(* CODESYS project traffic lights.project

Project tree, tasks and I/O mapping:
  Device : CODESYS Control Win V3, 3S - Smart Software Solutions GmbH, order no. 305021, version 3.5.7.0
    application Application
      libraries: Standard, * (System)
      task MainTask (cyclic, interval t#20ms, priority 1) calls PLC_PRG
      task VISU_TASK (cyclic, interval 100 ms, priority 31) calls VisuElems.Visu_Prg
      program PLC_PRG [LD]
      visualisation Visualization
  text list GlobalTextList
*)

// Device/Application/PLC_PRG
PROGRAM PLC_PRG

VAR
	TON_01: TON;
	t1: TIME;
	TP_01: TP;
	t11: TIME;
	F_TRIG_02: F_TRIG;
	TON_02: TON;
	t2: TIME;
	TP_02: TP;
	t22: TIME;
	F_TRIG_03: F_TRIG;
	F_TRIG_04: F_TRIG;
	TP_03: TP;
	TP_04: TP;
	t3: TIME;
	start: BOOL;
	stop: BOOL;
	lamp4: BOOL;
	lamp1: BOOL;
	lamp2: BOOL;
	lamp3: BOOL;
	red: BOOL;
	green: BOOL;
	amber: BOOL;
END_VAR

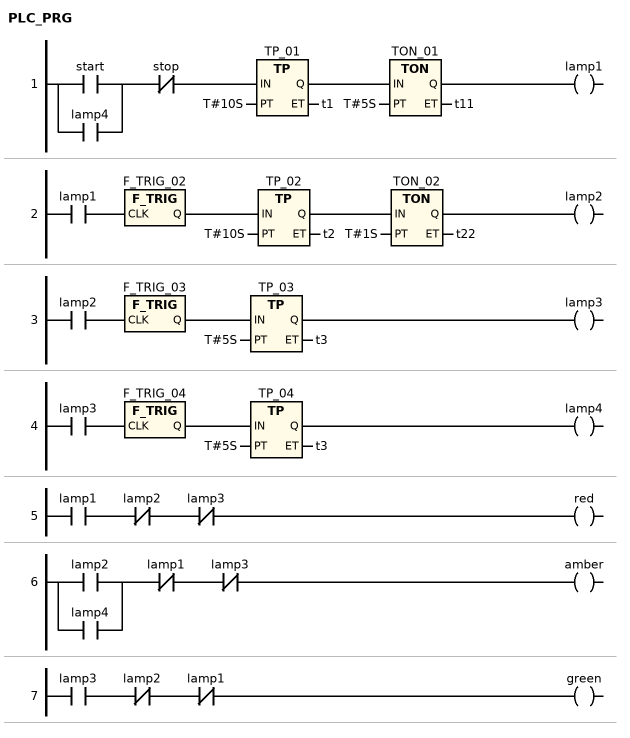
// NETWORK 1
TP_01(IN := (start OR lamp4) AND NOT stop, PT := T#10S, ET => t1); // TP
TON_01(IN := TP_01.Q, PT := T#5S, ET => t11); // TON
lamp1 := TON_01.Q;

// NETWORK 2
F_TRIG_02(CLK := lamp1); // F_TRIG
TP_02(IN := F_TRIG_02.Q, PT := T#10S, ET => t2); // TP
TON_02(IN := TP_02.Q, PT := T#1S, ET => t22); // TON
lamp2 := TON_02.Q;

// NETWORK 3
F_TRIG_03(CLK := lamp2); // F_TRIG
TP_03(IN := F_TRIG_03.Q, PT := T#5S, ET => t3); // TP
lamp3 := TP_03.Q;

// NETWORK 4
F_TRIG_04(CLK := lamp3); // F_TRIG
TP_04(IN := F_TRIG_04.Q, PT := T#5S, ET => t3); // TP
lamp4 := TP_04.Q;

// NETWORK 5
red := lamp1 AND NOT lamp2 AND NOT lamp3;

// NETWORK 6
amber := (lamp2 OR lamp4) AND NOT lamp1 AND NOT lamp3;

// NETWORK 7
green := lamp3 AND NOT lamp2 AND NOT lamp1;

END_PROGRAM

// Device/Application/Visualization
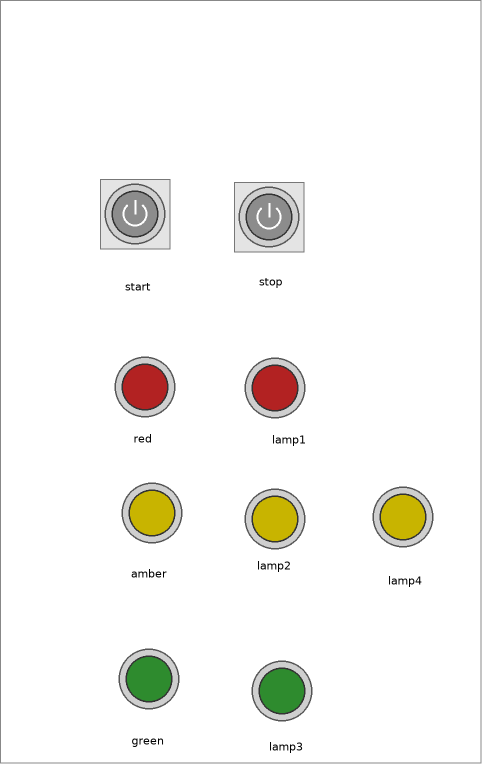
VISUALIZATION Visualization  // 482x764
    Lamp1 (110,352 70x70), variable: PLC_PRG.red, style: Lamp-Lamp1-Red
    Lamp1 (117,478 70x70), variable: PLC_PRG.amber, style: Lamp-Lamp1-Yellow
    Lamp1 (114,644 70x70), variable: PLC_PRG.green, style: Lamp-Lamp1-Green
    Lamp1 (240,484 70x70), variable: PLC_PRG.lamp2, style: Lamp-Lamp1-Yellow
    Lamp1 (368,482 70x70), variable: PLC_PRG.lamp4, style: Lamp-Lamp1-Yellow
    Lamp1 (240,353 70x70), variable: PLC_PRG.lamp1, style: Lamp-Lamp1-Red
    Lamp1 (247,656 70x70), variable: PLC_PRG.lamp3, style: Lamp-Lamp1-Green
    PowerSwitch (100,179 70x70), variable: PLC_PRG.start, behaviour: TOGGLE, style: Switch-PowerSwitch-Gray
    PowerSwitch (234,182 70x70), variable: PLC_PRG.stop, behaviour: TOGGLE, style: Switch-PowerSwitch-Gray
    Label (63,272 150x30), "start"
    Label (196,267 150x30), "stop"
    Label (68,424 150x30), "red"
    Label (214,425 150x30), "lamp1"
    Label (199,551 150x30), "lamp2"
    Label (74,559 150x30), "amber"
    Label (330,566 150x30), "lamp4"
    Label (73,726 150x30), "green"
    Label (211,732 150x30), "lamp3"
END_VISUALIZATION
